FUNCTION_BLOCK FB_Inverter
VAR_INPUT
END_VAR
VAR_OUTPUT
END_VAR
VAR
END_VAR

END_FUNCTION_BLOCK

(* stored: Version 1.1.0.1
   POU FB_Inverter: Id {48cb2406-29c9-4ea5-ad3e-84a50ffa6fc5}, SpecialFunc None *)
